// TIA Portal V18 export
TYPE "LGasp_type_impilaggio"
// stored: IsFailsafeCompliant false
   STRUCT
      nomeprogramma : WString[30];   // nome del programma trasferito dal PC
      ID : DInt;   // ID programma
      Tipoimpilaggio : DInt;   // 1= colonne affiancate 2= colonne sormontate 3 = ...
      DeltaX : LReal;   // [mm] incremento in X fra colonne adiacenti
      DeltaY : LReal;   // [mm] incremento in Y fra colonne adiacenti (solo in caso di colonne in 2 dimensioni)
      DeltaZ : LReal;   // [mm] incremento in Z fra righe adiacenti
      NrPzMaxPacco : DInt;   // Numero massimo di pezzi del pacco
      X_MaxPacco : LReal;   // [mm] Larghezza X massima del pacco
      Y_MaxPacco : LReal;   // [mm] Larghezza Y massima del pacco (solo in caso di colonne in 2 dimensioni)
      Z_MaxPacco : LReal;   // [mm] Altezza Z massima del pacco
      PesoTotMaxPacco : LReal;   // [kg] Peso totale massimo del pacco
      PesoLineareMaxPacco : LReal;   // [kg/m] Peso massimo del pacco per metro di lunghezza (opzionale)
   END_STRUCT;
END_TYPE
